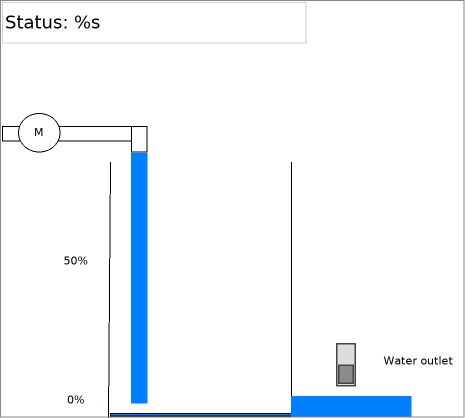
VISUALIZATION Visualization  // 465x418
    RoundedRectangle (110,413 182x3)
        p2773130477: - MAIN.mwTankLevel
    Textfield (2,2 304x41), "Status: %s", text variable: GVL.isStatusText
    Line (291,162) (291,415)
    Line (110,162) (108,418)
    Rectangle (2,126 145x15)
    Rectangle (131,126 16x26)
    Ellipse (18,113 42x39), "M"
    Rectangle (131,153 16x250), invisible if: Not MAIN.mxPumpOn
    Rectangle (291,396 120x20), invisible if: Not Main.mxOpenDrainingValve
    DipSwitch (318,343 56x43), variable: MAIN.mxOpenDrainingValve, behaviour: TOGGLE, style: Switch-DipSwitch-Gray
    Label (48,243 56x36), "50%"
    Label (48,382 56x36), "0%"
    Label (372,343 93x36), "Water outlet"
END_VISUALIZATION

(* stored: Version 1.1.0.1
   Visu Visualization: Id {291e9a6c-eb04-4490-b2e8-77faa3a8d12e} *)
